TYPE ST_HnhtHnltLinkageControl :
STRUCT
	fTargetTemperature_HNHT : REAL;
	fTargetTemperature_HNLT : REAL;
	bAlgorithmPermission_HNHT : BOOL;
	bAlgorithmPermission_HNLT : BOOL;
END_STRUCT
END_TYPE

(* stored: Version 1.1.0.1, ProductVersion 3.1.4024.10
   DUT ST_HnhtHnltLinkageControl: Id {885711f9-5e9c-420d-93f7-37d68a3b8222} *)
